// TIA Portal V18 export
TYPE "PLCtoMES_MainCheckOutStation1ST350_ext"
// stored: IsFailsafeCompliant false
   STRUCT
      CheckSum : Int;   // 校验和
      PartTypeID : Int;   // 产品类型
      PartTypeSN : String[60];   // 产品主体码
      PalletID : Int;
      PartStatus : Int;   // 产品加工结果（1 OK;2 NG）
      SubPartSN : String[60];   // 产品组件码
      StatusBits2 : DInt;   // 备用
      "PLCTransfer time" : String[60];   // 工位1作业时间日期
      DataMatrixStr : String[60];   // 打标二维码内容
      ProductNameStr : String[60];   // 打标产品名称
      HW_Str : String[60];   // 打标HW内容
      SW_Str : String[60];   // 打标SW内容
      PN_Str : String[60];   // 打标PN内容
      DATA_Str : String[60];   // 打标DATA内容
      SN_Str : String[60];   // 打标SN内容
      ECU_UID_Str : String[60];   // 打标ECU UID内容
      Vdc_Str : String[60];   // 打标电压内容
      Power_Str : String[60];   // 打标功率内容
      Place_Str : String[60];   // 打标产地内容
      Spare : Array[880..998] of Byte;   // 备用
      Massage : "PLCtoMES_AlarmMassage_ext";
   END_STRUCT;
END_TYPE
